(* PLC project Unnamed, Unknown Unnamed 1 *)
(* stored: creationDateTime 2013-01-29T14:01:00, modificationDateTime 2017-06-08T15:59:13 *)

(* Gets time in us from power up *)
FUNCTION US_TIME : UDINT
  VAR_INPUT
    NO_MATTER : INT;
  END_VAR

                        
                     {{
                     #include <stdint.h>
                     typedef uint32_t u32;
                     extern u32 getUsTimt (void);
                     US_TIME = getUsTimt();
                     }}
                    
                    
END_FUNCTION
